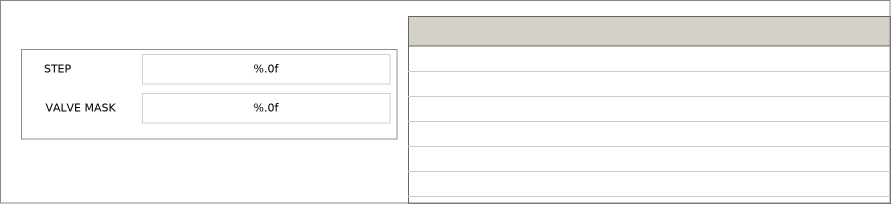
VISUALIZATION visControl  // 891x204
    Table (408,16 483x188), data array: GVL_visVariableMap.anValveMask
        p3854506369: GVL_visVariableMap.anValveMask[INDEX]
    Group (21,41 376x98)
        Group (7,13 362x69)
            Textfield (114,0 248x30), "%.0f", text variable: GVL_visVariableMap.visValveMaskIdx
                OnMouseClick: write GVL_visVariableMap.visValveMaskIdx via VisuDialogs.Numpad
            Textfield (114,39 248x30), "%.0f", text variable: GVL_visVariableMap.nValveMask
                OnMouseClick: write GVL_visVariableMap.nValveMask via VisuDialogs.Numpad
            Label (0,0 59x30), "STEP"
            Label (0,39 105x30), "VALVE MASK"
        GroupBox (0,0 376x98)
END_VISUALIZATION

(* stored: Version 1.1.0.1
   Visu visControl: Id {8f176c85-1c5d-0b37-0be5-b4c46381287b} *)
